ABB RobotStudio station: 实验一.rspag

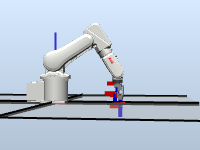
--- station ---
Station PartC (saved by RobotStudio 6.8.8148.134)
Controller System2
  mechanical unit ROB_1: IRB120_3_58__01, 6 joints, base frame (0, 0, 0) mm
Layout (positions relative to the parent item):
  - IRB120_3_58__01 [mechanism, from Robots\IRB120_3_58_G_01.rslib] at (0, 0, 0) mm; joint values [0.0862, 1.0205, 0.0168, -0.0598, 0.5437, 0.1489] (rad or m)
  - SmartComponent_1 [smart component] at (441.85, 35.96, 134.79) mm, rotated rx -178.18 ry -0.37 rz 179.34 deg
      signals: DI GET, DO FINISH
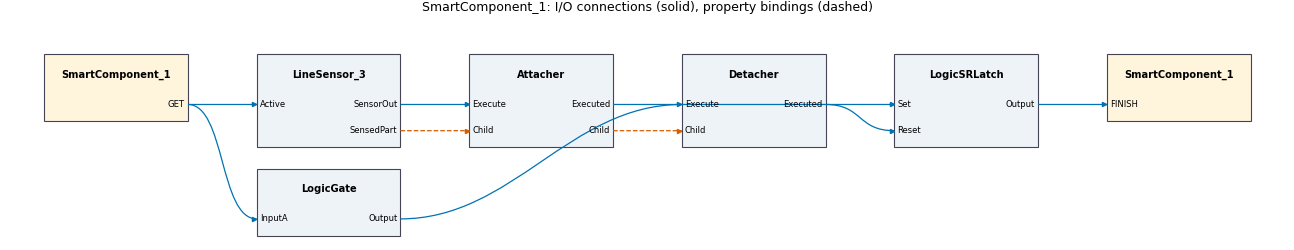
      connections:
        SmartComponent_1.GET -> LineSensor_3.Active
        SmartComponent_1.GET -> LogicGate.InputA
        LineSensor_3.SensorOut -> Attacher.Execute
        LogicGate.Output -> Detacher.Execute
        Attacher.Executed -> LogicSRLatch.Set
        Detacher.Executed -> LogicSRLatch.Reset
        LogicSRLatch.Output -> SmartComponent_1.FINISH
        LineSensor_3.SensedPart => Attacher.Child
        Attacher.Child => Detacher.Child
    - LineSensor_3 [smart component, from Components\LineSensor.rslib] at (-22.5, 0, 83.55) mm
        properties: Start=[0.0149998126219963 4.21158825841816E-07 0.0127464790726794]; End=[-0.0179682331662568 -0.0125006377603764 0.00370705963323065]; Radius=0.005; SensedPart=部件_2; SensedPoint=[0.450000061035156 0.0323275299072266 0.0388537902832031]
      - _sensorPart_ [part]
    - Attacher [smart component, from Components\Attacher.rslib]
        properties: Parent=SmartComponent_1; Flange=0; Child=部件_2; Mount=false; Offset=[0 0 0]; Orientation=[0 0 0]
    - Detacher [smart component, from Components\Detacher.rslib]
        properties: Child=部件_2; KeepPosition=true
    - LogicGate [smart component, from Components\LogicGate.rslib]
        properties: Operator=NOT; Delay=0
    - LogicSRLatch [smart component, from Components\LogicSRLatch.rslib]
    - My_Mechanism [mechanism] at (0, 0, 0) mm; joint values [0] (rad or m)
        TCP tool1 at (15.5, 0, 69.3) mm
        TCP tool2 at (-22.5, 0, 83.55) mm
        TCP tool3 at (-22.5, 0, 160.55) mm
        links: L1, L2
  - 部件_2 [part] at (0, 0, 23.06) mm
  - 框架_1 [frame] at (15.5, 0, 69.3) mm
  - 框架_2 [frame] at (-22.5, 0, 83.55) mm
  - 框架_3 [frame] at (-22.5, 0, 160.55) mm
Attachment: My_Mechanism is attached to IRB120_3_58__01 / Link6
Attachment: SmartComponent_1 is attached to IRB120_3_58__01 / Link6
Attachment: LineSensor_3 is attached to My_Mechanism / L1
Attachment: 部件_2 is attached to SmartComponent_1
EventTableEntry 2443: Group=, Trigger=DO_007 2444, Actions=[EventTableActionMechanicalPose 2445], Comment=, ActivationMode=2, Cyclic=false
EventTableTriggerIO 2444: IOValue=[1], IRC5Controller=? -1, Operator=0, SignalSource=System2 2451
EventTableActionMechanicalPose 2445: VirtualSignal=, Mechanism=My_Mechanism 980, ToPoseName=SyncPosition, VirtualSignalValue=[1]
EventTableEntry 2446: Group=, Trigger=DO_007 2447, Actions=[EventTableActionMechanicalPose 2448], Comment=, ActivationMode=2, Cyclic=false
EventTableTriggerIO 2447: IOValue=[0], IRC5Controller=? -1, Operator=0, SignalSource=System2 2451
EventTableActionMechanicalPose 2448: VirtualSignal=, Mechanism=My_Mechanism 980, ToPoseName=HomePosition, VirtualSignalValue=[1]
Station logic (signal -> signal, property => property):
  System2.DO_007 -> SmartComponent_1.GET
Targets, tools, work objects and paths stored in the station and not in the controller backup, written as RAPID:
! task T_ROB1
MODULE CalibData
  PERS tooldata tool1:=[TRUE,[[15.5,0,69.3],[1,0,0,0]],[1,[0,0,1],[1,0,0,0],0,0,0]];
  PERS tooldata tool2:=[TRUE,[[-22.5,0,83.554],[1,0,0,0]],[1,[0,0,1],[1,0,0,0],0,0,0]];
  PERS tooldata tool3:=[TRUE,[[-22.5,0,160.554],[1,0,0,0]],[1,[0,0,1],[1,0,0,0],0,0,0]];
  PERS tooldata Tooldata_4:=[TRUE,[[15.5,0,69.3],[1,0,0,0]],[1,[0,0,1],[1,0,0,0],0,0,0]];
  PERS tooldata Tooldata_5:=[TRUE,[[-22.5,0,83.554],[1,0,0,0]],[1,[0,0,1],[1,0,0,0],0,0,0]];
  PERS tooldata Tooldata_6:=[TRUE,[[-22.5,0,160.554],[1,0,0,0]],[1,[0,0,1],[1,0,0,0],0,0,0]];
ENDMODULE


--- Backups/System2/RAPID/TASK1/PROGMOD/Module1.mod ---
MODULE Module1
    !***********************************************************
    !
    ! Module:  Module1
    !
    ! Description:
    !   <Insert description here>
    !
    ! Author: He
    !
    ! Version: 1.0
    !
    !***********************************************************


    !***********************************************************
    !
    ! Procedure main
    !
    !   This is the entry point of your program
    !
    !***********************************************************
    PROC main()
        !Add your code here
    ENDPROC
ENDMODULE

--- Backups/System2/SYSPAR/EIO.cfg ---
EIO:CFG_1.0:6:1::
#
INDUSTRIAL_NETWORK:

      -Name "DeviceNet" -Label "DeviceNet Master/Slave Network" -Address "2"
#
DEVICENET_DEVICE:

      -Name "d652" -VendorName "ABB Robotics" -ProductName "24 VDC I/O Device"\
      -Label "DSQC 652 24 VDC I/O Device" -Address 10 -ProductCode 26\
      -DeviceType 7 -ConnectionType "COS" -OutputSize 2 -InputSize 2
#
DEVICENET_INTERNAL_DEVICE:

      -Name "DN_Internal_Device" -VendorName "ABB Robotics"\
      -ProductName "DeviceNet Internal Slave Device"
#
EIO_SIGNAL:

      -Name "DO_007" -SignalType "DO" -Device "d652" -DeviceMap "7"
